ABB RobotStudio station: Third  Behaviour.rspag

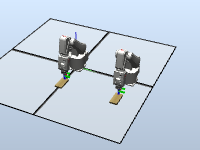
--- station ---
Station Station (saved by RobotStudio 6.8.8307.1040)
Controller Robot2, task T_ROB1: task frame (RAPID world) sits at (0, 700, 0) mm in the station
Controller Robot1
  mechanical unit ROB_1: IRB120_3_58__01, 6 joints, base frame (0, 0, 0) mm
Controller Robot2
  mechanical unit ROB_1: IRB120_3_58__01_2, 6 joints, base frame (0, 0, 0) mm
Layout (positions relative to the parent item):
  - IRB120_3_58__01 [mechanism, from Robots\IRB120_3_58_G_01.rslib] at (0, 0, 0) mm; joint values [0, 0.8108, 0.5752, 0, 0.1848, 0] (rad or m)
  - IRB120_3_58__01_2 [mechanism, from Robots\IRB120_3_58_G_01.rslib] at (0, 700, 0) mm; joint values [0, 0.8108, 0.5752, 0, 0.1848, 0] (rad or m)
  - Gripper [mechanism, from Libraries\Gripper.rslib] at (320, 0, 120) mm, rotated rx 180 ry 0 rz 180 deg
  - Gripper_2 [mechanism, from Libraries\Gripper.rslib] at (320, 700, 120) mm, rotated rx 180 ry 0 rz 180 deg
  - Pieza_1 [part] at (300, -45, 0) mm
  - Pieza_2 [part] at (330, -45, 0) mm
  - Pieza_3 [part] at (360, -45, 0) mm
  - Pieza_4 [part] at (390, -45, 0) mm
  - Pieza_5 [part] at (420, -45, 0) mm
  - Pieza_6 [part] at (450, -45, 0) mm
  - Pieza_7 [part] at (0, 700, 0) mm
  - Pieza_8 [part] at (0, 700, 0) mm
  - Pieza_9 [part] at (0, 700, 0) mm
  - Pieza_10 [part] at (0, 700, 0) mm
  - Pieza_11 [part] at (0, 700, 0) mm
  - Pieza_12 [part] at (0, 700, 0) mm
  - Grupo_3 [graphiccomponentgroup] at (0, 350, 0) mm
    - Pieza_11 [part] at (300, -45, 0) mm
    - Pieza_12 [part] at (330, -45, 0) mm
    - Pieza_13 [part] at (360, -45, 0) mm
    - Pieza_21 [part] at (390, -45, 20) mm, rotated rx 0 ry 0 rz 90 deg
    - Pieza_22 [part] at (390, -15, 20) mm, rotated rx 0 ry 0 rz 90 deg
    - Pieza_23 [part] at (390, 15, 20) mm, rotated rx 0 ry 0 rz 90 deg
    - Pieza_31 [part] at (300, -45, 40) mm
    - Pieza_32 [part] at (330, -45, 40) mm
    - Pieza_33 [part] at (360, -45, 40) mm
    - Pieza_41 [part] at (390, 15, 60) mm, rotated rx 0 ry 0 rz 90 deg
    - Pieza_42 [part] at (390, -15, 60) mm, rotated rx 0 ry 0 rz 90 deg
    - Pieza_43 [part] at (390, -45, 60) mm, rotated rx 0 ry 0 rz 90 deg
  - Attacher [smart component, from Components\Attacher.rslib]
      properties: Parent=Gripper; Flange=0; Child=Pieza_1; Mount=false; Offset=[0 0 0.01]; Orientation=[0 0 0]
  - Detacher [smart component, from Components\Detacher.rslib]
      properties: Child=Pieza_1; KeepPosition=true
  - Attacher_2 [smart component, from Components\Attacher.rslib]
      properties: Parent=Gripper; Flange=0; Child=Pieza_2; Mount=false; Offset=[0 0 0.01]; Orientation=[0 0 0]
  - Attacher_3 [smart component, from Components\Attacher.rslib]
      properties: Parent=Gripper; Flange=0; Child=Pieza_3; Mount=false; Offset=[0 0 0.01]; Orientation=[0 0 0]
  - Attacher_4 [smart component, from Components\Attacher.rslib]
      properties: Parent=Gripper; Flange=0; Child=Pieza_4; Mount=false; Offset=[0 0 0.01]; Orientation=[0 0 0]
  - Attacher_5 [smart component, from Components\Attacher.rslib]
      properties: Parent=Gripper; Flange=0; Child=Pieza_5; Mount=false; Offset=[0 0 0.01]; Orientation=[0 0 0]
  - Attacher_6 [smart component, from Components\Attacher.rslib]
      properties: Parent=Gripper; Flange=0; Child=Pieza_6; Mount=false; Offset=[0 0 0.01]; Orientation=[0 0 0]
  - Attacher_7 [smart component, from Components\Attacher.rslib]
      properties: Parent=Gripper_2; Flange=0; Child=Pieza_7; Mount=false; Offset=[0 0 0.01]; Orientation=[0 0 0]
  - Detacher_2 [smart component, from Components\Detacher.rslib]
      properties: Child=Pieza_2; KeepPosition=true
  - Detacher_3 [smart component, from Components\Detacher.rslib]
      properties: Child=Pieza_3; KeepPosition=true
  - Detacher_4 [smart component, from Components\Detacher.rslib]
      properties: Child=Pieza_4; KeepPosition=true
  - Detacher_5 [smart component, from Components\Detacher.rslib]
      properties: Child=Pieza_5; KeepPosition=true
  - Detacher_6 [smart component, from Components\Detacher.rslib]
      properties: Child=Pieza_6; KeepPosition=true
  - Attacher_8 [smart component, from Components\Attacher.rslib]
      properties: Parent=Gripper_2; Flange=0; Child=Pieza_8; Mount=false; Offset=[0 0 0.01]; Orientation=[0 0 0]
  - Attacher_9 [smart component, from Components\Attacher.rslib]
      properties: Parent=Gripper_2; Flange=0; Child=Pieza_9; Mount=false; Offset=[0 0 0.01]; Orientation=[0 0 0]
  - Attacher_10 [smart component, from Components\Attacher.rslib]
      properties: Parent=Gripper_2; Flange=0; Child=Pieza_10; Mount=false; Offset=[0 0 0.01]; Orientation=[0 0 0]
  - Attacher_11 [smart component, from Components\Attacher.rslib]
      properties: Parent=Gripper_2; Flange=0; Child=Pieza_11; Mount=false; Offset=[0 0 0.01]; Orientation=[0 0 0]
  - Attacher_12 [smart component, from Components\Attacher.rslib]
      properties: Parent=Gripper_2; Flange=0; Child=Pieza_12; Mount=false; Offset=[0 0 0.01]; Orientation=[0 0 0]
  - Detacher_7 [smart component, from Components\Detacher.rslib]
      properties: Child=Pieza_7; KeepPosition=true
  - Detacher_8 [smart component, from Components\Detacher.rslib]
      properties: Child=Pieza_8; KeepPosition=true
  - Detacher_9 [smart component, from Components\Detacher.rslib]
      properties: Child=Pieza_9; KeepPosition=true
  - Detacher_10 [smart component, from Components\Detacher.rslib]
      properties: Child=Pieza_10; KeepPosition=true
  - Detacher_11 [smart component, from Components\Detacher.rslib]
      properties: Child=Pieza_11; KeepPosition=true
  - Detacher_12 [smart component, from Components\Detacher.rslib]
      properties: Child=Pieza_12; KeepPosition=true
Attachment: Gripper is attached to IRB120_3_58__01 / Link6
Attachment: Gripper_2 is attached to IRB120_3_58__01_2 / Link6
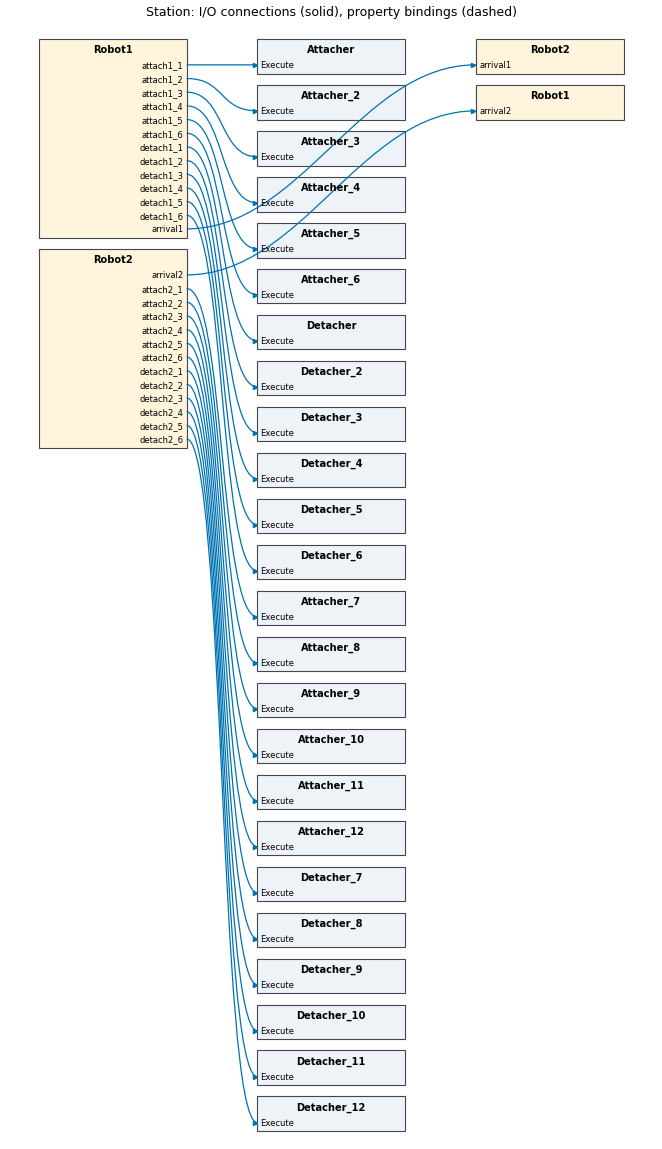
Station logic (signal -> signal, property => property):
  Robot1.attach1_1 -> Attacher.Execute
  Robot1.attach1_2 -> Attacher_2.Execute
  Robot1.attach1_3 -> Attacher_3.Execute
  Robot1.attach1_4 -> Attacher_4.Execute
  Robot1.attach1_5 -> Attacher_5.Execute
  Robot1.attach1_6 -> Attacher_6.Execute
  Robot1.detach1_1 -> Detacher.Execute
  Robot1.detach1_2 -> Detacher_2.Execute
  Robot1.detach1_3 -> Detacher_3.Execute
  Robot1.detach1_4 -> Detacher_4.Execute
  Robot1.detach1_5 -> Detacher_5.Execute
  Robot1.detach1_6 -> Detacher_6.Execute
  Robot1.arrival1 -> Robot2.arrival1
  Robot2.arrival2 -> Robot1.arrival2
  Robot2.attach2_1 -> Attacher_7.Execute
  Robot2.attach2_2 -> Attacher_8.Execute
  Robot2.attach2_3 -> Attacher_9.Execute
  Robot2.attach2_4 -> Attacher_10.Execute
  Robot2.attach2_5 -> Attacher_11.Execute
  Robot2.attach2_6 -> Attacher_12.Execute
  Robot2.detach2_1 -> Detacher_7.Execute
  Robot2.detach2_2 -> Detacher_8.Execute
  Robot2.detach2_3 -> Detacher_9.Execute
  Robot2.detach2_4 -> Detacher_10.Execute
  Robot2.detach2_5 -> Detacher_11.Execute
  Robot2.detach2_6 -> Detacher_12.Execute

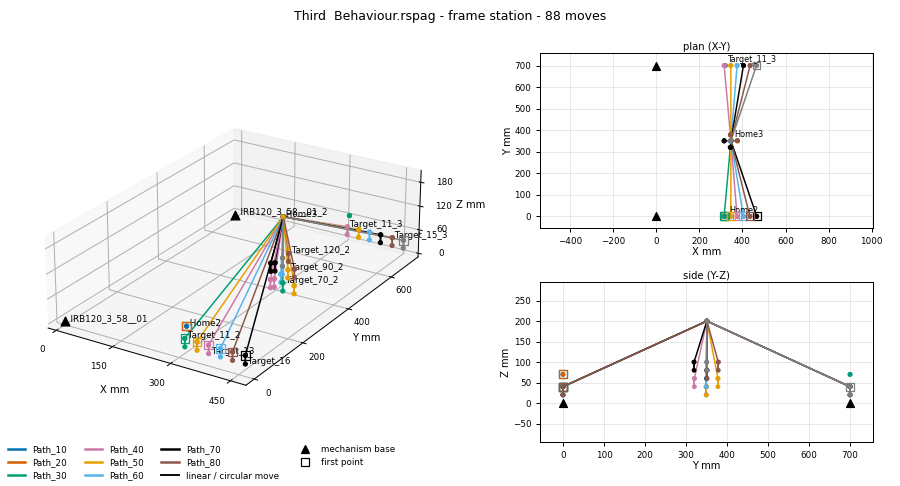
[picture p0: tool path of Third  Behaviour.rspag in frame station, 88 of 88 moves have a stored position in this frame; points joined in program order, loops and branches not executed]
--- Backups/Robot1/RAPID/TASK1/PROGMOD/CalibData.mod ---
MODULE CalibData
	PERS tooldata Gripper:=[TRUE,[[0,0,50],[1,0,0,0]],[1,[0,0,1],[1,0,0,0],0,0,0]];
ENDMODULE

--- Backups/Robot1/RAPID/TASK1/PROGMOD/Module1.mod ---
MODULE Module1
	CONST robtarget Home:=[[407.655099262,0,569],[0.5,0,0.866025404,0],[0,0,0,0],[9E+09,9E+09,9E+09,9E+09,9E+09,9E+09]];
    CONST robtarget Home2:=[[320,0,70],[0,0,1,0],[0,0,0,0],[9E+09,9E+09,9E+09,9E+09,9E+09,9E+09]];
    CONST robtarget Home3:=[[346.394,350.952,200],[0,0,1,0],[0,0,0,0],[9E+09,9E+09,9E+09,9E+09,9E+09,9E+09]];
    CONST robtarget Target_11_2:=[[315,0,40],[0,0,1,0],[0,0,0,0],[9E+09,9E+09,9E+09,9E+09,9E+09,9E+09]];
    CONST robtarget Target_11:=[[315,0,20],[0,0,1,0],[0,0,0,0],[9E+09,9E+09,9E+09,9E+09,9E+09,9E+09]];
    CONST robtarget Target_70_2:=[[347.529,349.304,40],[0,0,1,0],[0,0,0,0],[9E+09,9E+09,9E+09,9E+09,9E+09,9E+09]];
    CONST robtarget Target_70:=[[347.529,349.304,20],[0,0,1,0],[0,0,0,0],[9E+09,9E+09,9E+09,9E+09,9E+09,9E+09]];
    CONST robtarget Target_12_2:=[[345.811,0,40],[0,0,1,0],[0,0,0,0],[9E+09,9E+09,9E+09,9E+09,9E+09,9E+09]];
    CONST robtarget Target_12:=[[345.811,0,20],[0,0,1,0],[0,0,0,0],[9E+09,9E+09,9E+09,9E+09,9E+09,9E+09]];
    CONST robtarget Target_80_2:=[[342.623,320.48,60],[0,0.707106781,0.707106781,0],[0,0,0,0],[9E+09,9E+09,9E+09,9E+09,9E+09,9E+09]];
    CONST robtarget Target_80:=[[342.623,320.48,40],[0,0.707106781,0.707106781,0],[0,0,0,0],[9E+09,9E+09,9E+09,9E+09,9E+09,9E+09]];
    CONST robtarget Target_13_2:=[[374.984,0,40],[0,0,1,0],[0,0,0,0],[9E+09,9E+09,9E+09,9E+09,9E+09,9E+09]];
    CONST robtarget Target_13:=[[374.984,0,20],[0,0,1,0],[0,0,0,0],[9E+09,9E+09,9E+09,9E+09,9E+09,9E+09]];
    CONST robtarget Target_90_2:=[[343.622,377.935,60],[0,0.707106781,0.707106781,0],[0,0,0,0],[9E+09,9E+09,9E+09,9E+09,9E+09,9E+09]];
    CONST robtarget Target_90:=[[343.622,377.935,40],[0,0.707106781,0.707106781,0],[0,0,0,0],[9E+09,9E+09,9E+09,9E+09,9E+09,9E+09]];
    CONST robtarget Target_14_2:=[[404.545,0,40],[0,0,1,0],[0,0,0,0],[9E+09,9E+09,9E+09,9E+09,9E+09,9E+09]];
    CONST robtarget Target_14:=[[404.545,0,20],[0,0,1,0],[0,0,0,0],[9E+09,9E+09,9E+09,9E+09,9E+09,9E+09]];
    CONST robtarget Target_100_2:=[[345.507,350.362,80],[0,0,1,0],[0,0,0,0],[9E+09,9E+09,9E+09,9E+09,9E+09,9E+09]];
    CONST robtarget Target_100:=[[345.507,350.362,60],[0,0,1,0],[0,0,0,0],[9E+09,9E+09,9E+09,9E+09,9E+09,9E+09]];
    CONST robtarget Target_15_2:=[[434.489,0,40],[0,0,1,0],[0,0,0,0],[9E+09,9E+09,9E+09,9E+09,9E+09,9E+09]];
    CONST robtarget Target_15:=[[434.489,0,20],[0,0,1,0],[0,0,0,0],[9E+09,9E+09,9E+09,9E+09,9E+09,9E+09]];
    CONST robtarget Target_110_2:=[[344.715,319.63,100],[0,0.707106781,0.707106781,0],[0,0,0,0],[9E+09,9E+09,9E+09,9E+09,9E+09,9E+09]];
    CONST robtarget Target_110:=[[344.715,319.63,80],[0,0.707106781,0.707106781,0],[0,0,0,0],[9E+09,9E+09,9E+09,9E+09,9E+09,9E+09]];
    CONST robtarget Target_16_2:=[[466.137,0,40],[0,0,1,0],[0,0,0,0],[9E+09,9E+09,9E+09,9E+09,9E+09,9E+09]];
    CONST robtarget Target_16:=[[466.137,0,20],[0,0,1,0],[0,0,0,0],[9E+09,9E+09,9E+09,9E+09,9E+09,9E+09]];
    CONST robtarget Target_120_2:=[[344.186,378.736,100],[0,0.707106781,0.707106781,0],[0,0,0,0],[9E+09,9E+09,9E+09,9E+09,9E+09,9E+09]];
    CONST robtarget Target_120:=[[344.186,378.736,80],[0,0.707106781,0.707106781,0],[0,0,0,0],[9E+09,9E+09,9E+09,9E+09,9E+09,9E+09]];
    !***********************************************************
    !
    ! Módulo:  Module1
    !
    ! Descripción:
    !   <Introduzca la descripción aquí>
    !
    ! Autor: Zuleika
    !
    ! Versión: 1.0
    !
    !***********************************************************


    !***********************************************************
    !
    ! Procedimiento Main
    !
    !   Este es el punto de entrada de su programa
    !
    !***********************************************************
    PROC main()
        SetDO arrival1, 0;

        Path_10;

        SetDo arrival1, 1;

        WaitDI arrival2, 1;
        SetDo arrival1, 0;

        Path_30;

        SetDO arrival1, 1;

        Path_20;

        SetDo arrival1, 0;
        WaitDI arrival2, 1;

        Path_50;

        SetDO arrival1, 1;

        Path_20;

        SetDo arrival1, 0;
        WaitDI arrival2, 1;

        Path_40;

        SetDO arrival1, 1;

        Path_20;

        SetDo arrival1, 0;
        WaitDI arrival2, 1;

        Path_60;

        SetDO arrival1, 1;

        Path_20;

        SetDo arrival1, 0;
        WaitDI arrival2, 1;

        Path_80;

        SetDO arrival1, 1;

        Path_20;

        SetDo arrival1, 0;
        WaitDI arrival2, 1;

        Path_70;

        SetDO arrival1, 1;

        Path_20;

        SetDo arrival1, 0;

        !PulseDO attach1_1;
        !WaitTime 1;
        !PulseDo detach1_1;
        !WaitTime 1;
    ENDPROC
	PROC Path_10()
        MoveL Home2,v300,z100,Gripper\WObj:=wobj0;
	ENDPROC
    PROC Path_20()
        MoveL Home2,v300,z100,Gripper\WObj:=wobj0;
    ENDPROC
    PROC Path_30()
        MoveL Target_11_2,v300,z0,Gripper\WObj:=wobj0;
        MoveL Target_11,v300,fine,Gripper\WObj:=wobj0;
        PulseDO attach1_1;
        WaitTime 1;
        MoveL Target_11_2,v300,z0,Gripper\WObj:=wobj0;
        MoveL Home3,v300,z0,Gripper\WObj:=wobj0;
        MoveL Target_70_2,v300,z0,Gripper\WObj:=wobj0;
        MoveL Target_70,v300,fine,Gripper\WObj:=wobj0;
        PulseDo detach1_1;
        WaitTime 1;
        MoveL Target_70_2,v300,z0,Gripper\WObj:=wobj0;
    ENDPROC
    PROC Path_40()
        MoveL Target_13_2,v300,z0,Gripper\WObj:=wobj0;
        MoveL Target_13,v300,fine,Gripper\WObj:=wobj0;
        PulseDO attach1_3;
        WaitTime 1;
        MoveL Target_13_2,v300,z0,Gripper\WObj:=wobj0;
        MoveL Home3,v300,z0,Gripper\WObj:=wobj0;
        MoveL Target_80_2,v300,z0,Gripper\WObj:=wobj0;
        MoveL Target_80,v300,fine,Gripper\WObj:=wobj0;
        PulseDo detach1_3;
        WaitTime 1;
        MoveL Target_80_2,v300,z0,Gripper\WObj:=wobj0;
    ENDPROC
    PROC Path_50()
        MoveL Target_12_2,v300,z0,Gripper\WObj:=wobj0;
        MoveL Target_12,v300,fine,Gripper\WObj:=wobj0;
        PulseDO attach1_2;
        WaitTime 1;
        MoveL Target_12_2,v300,z0,Gripper\WObj:=wobj0;
        MoveL Home3,v300,z0,Gripper\WObj:=wobj0;
        MoveL Target_90_2,v300,z0,Gripper\WObj:=wobj0;
        MoveL Target_90,v300,fine,Gripper\WObj:=wobj0;
        PulseDo detach1_2;
        WaitTime 1;
        MoveL Target_90_2,v300,z0,Gripper\WObj:=wobj0;
    ENDPROC
    PROC Path_60()
        MoveL Target_14_2,v300,z0,Gripper\WObj:=wobj0;
        MoveL Target_14,v300,fine,Gripper\WObj:=wobj0;
        PulseDO attach1_4;
        WaitTime 1;
        MoveL Target_14_2,v300,z0,Gripper\WObj:=wobj0;
        MoveL Home3,v300,z0,Gripper\WObj:=wobj0;
        MoveL Target_100_2,v300,z0,Gripper\WObj:=wobj0;
        MoveL Target_100,v300,fine,Gripper\WObj:=wobj0;
        PulseDo detach1_4;
        WaitTime 1;
        MoveL Target_100_2,v300,z0,Gripper\WObj:=wobj0;
    ENDPROC
    PROC Path_70()
        MoveL Target_16_2,v300,z0,Gripper\WObj:=wobj0;
        MoveL Target_16,v300,fine,Gripper\WObj:=wobj0;
        PulseDO attach1_6;
        WaitTime 1;
        MoveL Target_16_2,v300,z0,Gripper\WObj:=wobj0;
        MoveL Home3,v300,z0,Gripper\WObj:=wobj0;
        MoveL Target_110_2,v300,z0,Gripper\WObj:=wobj0;
        MoveL Target_110,v300,fine,Gripper\WObj:=wobj0;
        PulseDo detach1_6;
        WaitTime 1;
        MoveL Target_110_2,v300,z0,Gripper\WObj:=wobj0;
    ENDPROC
    PROC Path_80()
        MoveL Target_15_2,v300,z0,Gripper\WObj:=wobj0;
        MoveL Target_15,v300,fine,Gripper\WObj:=wobj0;
        PulseDO attach1_5;
        WaitTime 1;
        MoveL Target_15_2,v300,z0,Gripper\WObj:=wobj0;
        MoveL Home3,v300,z0,Gripper\WObj:=wobj0;
        MoveL Target_120_2,v300,z0,Gripper\WObj:=wobj0;
        MoveL Target_120,v300,fine,Gripper\WObj:=wobj0;
        PulseDo detach1_5;
        WaitTime 1;
        MoveL Target_120_2,v300,z0,Gripper\WObj:=wobj0;
    ENDPROC
ENDMODULE

--- Backups/Robot2/RAPID/TASK1/PROGMOD/Module1.mod ---
MODULE Module1
	CONST robtarget Home:=[[407.655099262,0,569],[0.353553391,0.612372436,0.612372436,0.353553391],[0,0,0,0],[9E+09,9E+09,9E+09,9E+09,9E+09,9E+09]];
    CONST robtarget Home2:=[[320,0,70],[0,0,1,0],[0,0,0,0],[9E+09,9E+09,9E+09,9E+09,9E+09,9E+09]];
    CONST robtarget Home3:=[[346.394,-349.048,200],[0,0,1,0],[0,0,0,0],[9E+09,9E+09,9E+09,9E+09,9E+09,9E+09]];
    CONST robtarget Target_11_3:=[[315,0,40],[0,0,1,0],[0,0,0,0],[9E+09,9E+09,9E+09,9E+09,9E+09,9E+09]];
    CONST robtarget Target_11:=[[315,0,20],[0,0,1,0],[0,0,0,0],[9E+09,9E+09,9E+09,9E+09,9E+09,9E+09]];
    CONST robtarget Target_70_3:=[[315.197,-350.536,40],[0,0,1,0],[0,0,0,0],[9E+09,9E+09,9E+09,9E+09,9E+09,9E+09]];
    CONST robtarget Target_70:=[[315.197,-350.536,20],[0,0,1,0],[0,0,0,0],[9E+09,9E+09,9E+09,9E+09,9E+09,9E+09]];
    CONST robtarget Target_12_3:=[[345.811,0,40],[0,0,1,0],[0,0,0,0],[9E+09,9E+09,9E+09,9E+09,9E+09,9E+09]];
    CONST robtarget Target_12:=[[345.811,0,20],[0,0,1,0],[0,0,0,0],[9E+09,9E+09,9E+09,9E+09,9E+09,9E+09]];
    CONST robtarget Target_80_3:=[[376.647,-350.123,40],[0,0,1,0],[0,0,0,0],[9E+09,9E+09,9E+09,9E+09,9E+09,9E+09]];
    CONST robtarget Target_80:=[[376.647,-350.123,20],[0,0,1,0],[0,0,0,0],[9E+09,9E+09,9E+09,9E+09,9E+09,9E+09]];
    CONST robtarget Target_13_3:=[[374.984,0,40],[0,0,1,0],[0,0,0,0],[9E+09,9E+09,9E+09,9E+09,9E+09,9E+09]];
    CONST robtarget Target_13:=[[374.984,0,20],[0,0,1,0],[0,0,0,0],[9E+09,9E+09,9E+09,9E+09,9E+09,9E+09]];
    CONST robtarget Target_90_3:=[[342.308,-350.408,60],[0,0.707106781,0.707106781,0],[0,0,0,0],[9E+09,9E+09,9E+09,9E+09,9E+09,9E+09]];
    CONST robtarget Target_90:=[[342.308,-350.408,40],[0,0.707106781,0.707106781,0],[0,0,0,0],[9E+09,9E+09,9E+09,9E+09,9E+09,9E+09]];
    CONST robtarget Target_14_3:=[[404.545,0,40],[0,0,1,0],[0,0,0,0],[9E+09,9E+09,9E+09,9E+09,9E+09,9E+09]];
    CONST robtarget Target_14:=[[404.545,0,20],[0,0,1,0],[0,0,0,0],[9E+09,9E+09,9E+09,9E+09,9E+09,9E+09]];
    CONST robtarget Target_100_3:=[[314.973,-349.258,80],[0,0,1,0],[0,0,0,0],[9E+09,9E+09,9E+09,9E+09,9E+09,9E+09]];
    CONST robtarget Target_100:=[[314.973,-349.258,60],[0,0,1,0],[0,0,0,0],[9E+09,9E+09,9E+09,9E+09,9E+09,9E+09]];
    CONST robtarget Target_15_3:=[[435.489,0,40],[0,0,1,0],[0,0,0,0],[9E+09,9E+09,9E+09,9E+09,9E+09,9E+09]];
    CONST robtarget Target_15:=[[435.489,0,20],[0,0,1,0],[0,0,0,0],[9E+09,9E+09,9E+09,9E+09,9E+09,9E+09]];
    CONST robtarget Target_110_3:=[[376.029,-348.718,80],[0,0,1,0],[0,0,0,0],[9E+09,9E+09,9E+09,9E+09,9E+09,9E+09]];
    CONST robtarget Target_110:=[[376.029,-348.718,60],[0,0,1,0],[0,0,0,0],[9E+09,9E+09,9E+09,9E+09,9E+09,9E+09]];
    CONST robtarget Target_16_3:=[[465.137,0,40],[0,0,1,0],[0,0,0,0],[9E+09,9E+09,9E+09,9E+09,9E+09,9E+09]];
    CONST robtarget Target_16:=[[465.137,0,20],[0,0,1,0],[0,0,0,0],[9E+09,9E+09,9E+09,9E+09,9E+09,9E+09]];
    CONST robtarget Target_120_3:=[[345.724,-349.521,100],[0,0.707106781,0.707106781,0],[0,0,0,0],[9E+09,9E+09,9E+09,9E+09,9E+09,9E+09]];
    CONST robtarget Target_120:=[[345.724,-349.521,80],[0,0.707106781,0.707106781,0],[0,0,0,0],[9E+09,9E+09,9E+09,9E+09,9E+09,9E+09]];
    !***********************************************************
    !
    ! Módulo:  Module1
    !
    ! Descripción:
    !   <Introduzca la descripción aquí>
    !
    ! Autor: Zuleika
    !
    ! Versión: 1.0
    !
    !***********************************************************


    !***********************************************************
    !
    ! Procedimiento Main
    !
    !   Este es el punto de entrada de su programa
    !
    !***********************************************************
    PROC main()
        SetDo arrival2, 0;

        Path_10;

        !SetDo arrival2, 1;

        WaitDI arrival1, 1;
        SetDo arrival2, 0;

        Path_40;

        SetDo arrival2, 1;

        Path_30;

        SetDo arrival2, 0;
        WaitDI arrival1, 1;

        Path_50;

        SetDo arrival2, 1;

        Path_30;

        SetDo arrival2, 0;
        WaitDI arrival1, 1;

        Path_60;

        SetDo arrival2, 1;

        Path_30;

        SetDo arrival2, 0;
        WaitDI arrival1, 1;

        Path_70;

        SetDo arrival2, 1;

        Path_30;

        SetDo arrival2, 0;
        WaitDI arrival1, 1;

        Path_80;

        SetDo arrival2, 1;

        Path_30;

        SetDo arrival2, 0;
        WaitDI arrival1, 1;

        Path_90;

        SetDo arrival2, 1;

        Path_30;

        SetDo arrival2, 0;

        !PulseDO attach2_1;
        !WaitTime 1;
        !PulseDO detach2_1;
        !WaitTime 1;
    ENDPROC
	PROC Path_10()
        MoveL Home2,v300,z100,Gripper\WObj:=wobj0;
	ENDPROC
    PROC Path_30()
        MoveL Home2,v300,z100,Gripper\WObj:=wobj0;
    ENDPROC
    PROC Path_40()
        MoveL Target_11_3,v300,z0,Gripper\WObj:=wobj0;
        MoveL Target_11,v300,fine,Gripper\WObj:=wobj0;
        PulseDO attach2_1;
        WaitTime 1;
        MoveL Target_11_3,v300,z0,Gripper\WObj:=wobj0;
        MoveL Home3,v300,z0,Gripper\WObj:=wobj0;
        MoveL Target_70_3,v300,z0,Gripper\WObj:=wobj0;
        MoveL Target_70,v300,fine,Gripper\WObj:=wobj0;
        PulseDO detach2_1;
        WaitTime 1;
        MoveL Target_70_3,v300,z0,Gripper\WObj:=wobj0;
    ENDPROC
    PROC Path_50()
        MoveL Target_12_3,v300,z0,Gripper\WObj:=wobj0;
        MoveL Target_12,v300,fine,Gripper\WObj:=wobj0;
        PulseDO attach2_2;
        WaitTime 1;
        MoveL Target_12_3,v300,z0,Gripper\WObj:=wobj0;
        MoveL Home3,v300,z0,Gripper\WObj:=wobj0;
        MoveL Target_80_3,v300,z0,Gripper\WObj:=wobj0;
        MoveL Target_80,v300,fine,Gripper\WObj:=wobj0;
        PulseDO detach2_2;
        WaitTime 1;
        MoveL Target_80_3,v300,z0,Gripper\WObj:=wobj0;
    ENDPROC
    PROC Path_60()
        MoveL Target_13_3,v300,z0,Gripper\WObj:=wobj0;
        MoveL Target_13,v300,fine,Gripper\WObj:=wobj0;
        PulseDO attach2_3;
        WaitTime 1;
        MoveL Target_13_3,v300,z0,Gripper\WObj:=wobj0;
        MoveL Home3,v300,z0,Gripper\WObj:=wobj0;
        MoveL Target_90_3,v300,z0,Gripper\WObj:=wobj0;
        MoveL Target_90,v300,fine,Gripper\WObj:=wobj0;
        PulseDO detach2_3;
        WaitTime 1;
        MoveL Target_90_3,v300,z0,Gripper\WObj:=wobj0;
    ENDPROC
    PROC Path_70()
        MoveL Target_14_3,v300,z0,Gripper\WObj:=wobj0;
        MoveL Target_14,v300,fine,Gripper\WObj:=wobj0;
        PulseDO attach2_4;
        WaitTime 1;
        MoveL Target_14_3,v300,z0,Gripper\WObj:=wobj0;
        MoveL Home3,v300,z0,Gripper\WObj:=wobj0;
        MoveL Target_100_3,v300,z0,Gripper\WObj:=wobj0;
        MoveL Target_100,v300,fine,Gripper\WObj:=wobj0;
        PulseDO detach2_4;
        WaitTime 1;
        MoveL Target_100_3,v300,z0,Gripper\WObj:=wobj0;
    ENDPROC
    PROC Path_80()
        MoveL Target_15_3,v300,z0,Gripper\WObj:=wobj0;
        MoveL Target_15,v300,fine,Gripper\WObj:=wobj0;
        PulseDO attach2_5;
        WaitTime 1;
        MoveL Target_15_3,v300,z0,Gripper\WObj:=wobj0;
        MoveL Home3,v300,z0,Gripper\WObj:=wobj0;
        MoveL Target_110_3,v300,z0,Gripper\WObj:=wobj0;
        MoveL Target_110,v300,fine,Gripper\WObj:=wobj0;
        PulseDO detach2_5;
        WaitTime 1;
        MoveL Target_110_3,v300,z0,Gripper\WObj:=wobj0;
    ENDPROC
    PROC Path_90()
        MoveL Target_16_3,v300,z0,Gripper\WObj:=wobj0;
        MoveL Target_16,v300,fine,Gripper\WObj:=wobj0;
        PulseDO attach2_6;
        WaitTime 1;
        MoveL Target_16_3,v300,z0,Gripper\WObj:=wobj0;
        MoveL Home3,v300,z0,Gripper\WObj:=wobj0;
        MoveL Target_120_3,v300,z0,Gripper\WObj:=wobj0;
        MoveL Target_120,v300,fine,Gripper\WObj:=wobj0;
        PulseDO detach2_6;
        WaitTime 1;
        MoveL Target_120_3,v300,z0,Gripper\WObj:=wobj0;
    ENDPROC
ENDMODULE

--- Backups/Robot1/SYSPAR/EIO.cfg ---
EIO:CFG_1.0:6:1::
#
EIO_SIGNAL:

      -Name "arrival1" -SignalType "DO"

      -Name "arrival2" -SignalType "DI"

      -Name "attach1_1" -SignalType "DO"

      -Name "attach1_2" -SignalType "DO"

      -Name "attach1_3" -SignalType "DO"

      -Name "attach1_4" -SignalType "DO"

      -Name "attach1_5" -SignalType "DO"

      -Name "attach1_6" -SignalType "DO"

      -Name "detach1_1" -SignalType "DO"

      -Name "detach1_2" -SignalType "DO"

      -Name "detach1_3" -SignalType "DO"

      -Name "detach1_4" -SignalType "DO"

      -Name "detach1_5" -SignalType "DO"

      -Name "detach1_6" -SignalType "DO"

--- Backups/Robot2/SYSPAR/EIO.cfg ---
EIO:CFG_1.0:6:1::
#
EIO_SIGNAL:

      -Name "arrival1" -SignalType "DI"

      -Name "arrival2" -SignalType "DO"

      -Name "attach2_1" -SignalType "DO"

      -Name "attach2_2" -SignalType "DO"

      -Name "attach2_3" -SignalType "DO"

      -Name "attach2_4" -SignalType "DO"

      -Name "attach2_5" -SignalType "DO"

      -Name "attach2_6" -SignalType "DO"

      -Name "detach2_1" -SignalType "DO"

      -Name "detach2_2" -SignalType "DO"

      -Name "detach2_3" -SignalType "DO"

      -Name "detach2_4" -SignalType "DO"

      -Name "detach2_5" -SignalType "DO"

      -Name "detach2_6" -SignalType "DO"
